(* CODESYS project connect_1.project
   Title: connect_1
   Version: 0.0.0.0
   Author: gusta

Project tree, tasks and I/O mapping:
  MyController : TM241CEC24T/U, Schneider Electric, order no. TM241CEC24T/U, version 4.0.6.18
    application Application
      libraries: Util, 3.5.1.0 (System)
      task MAST (cyclic, interval t#20ms, priority 15) calls opstart
      task Task (cyclic, interval t#5ms, priority 1) calls loop1
      task Task_1 (cyclic, interval t#20ms, priority 3) calls counter
      global variables GVL
      program opstart [ST]
      program counter [ST]
      program loop1 [ST]
      function block GPID [ST]
      program POU_1 [FBD]
    DI : Digital Inputs, Schneider Electric, version 4.0.6.18
        settings: IOs Usage = 15
        input  Application.input1 : BOOL  // IW0.I4
        input  Application.input2 : BOOL  // IW0.I5
        input  ibDI_IB1 : BYTE  // IB1
        unmapped channels: IW0
    DQ : Digital Outputs, Schneider Electric, version 4.0.6.18
        output Application.Q_enable : BOOL  // QW0.Q0
        output Application.Q_reset : BOOL  // QW0.Q1
        output Application.Q_operating : BOOL  // QW0.Q2
        output qbDQ_QB1 : BYTE  // QB1
        unmapped channels: QW0
    Counters : Counters, Schneider Electric, version 4.0.6.18
        settings: Instance name = 'HSCS'; B input History = 'old=-1 new=1'; A input History = 'old=-1 new=0'; Temporary Instance name = 'HSCS'; Instance name = 'HSCM'; B input History = 'old=-1 new=3'; A input History = 'old=-1 new=2'; Temporary Instance name = 'HSCM'
    Pulse_Generators : Pulse Generators, Schneider Electric, version 4.0.6.18
    Cartridge_1 : Cartridge, Schneider Electric, version 4.0.6.18
    IO_Bus : IO bus - TM3, Schneider Electric, version 4.0.6.18
      Module_1 : TM3AQ4/G, Schneider Electric, order no. TM3AQ4/G, version 1.0.0.12
          settings: KPI Configuration.KPI Configuration[0] = 17; KPI Configuration.KPI Configuration[1] = 17; KPI Configuration.KPI Configuration[4] = 240; KPI Configuration.KPI Configuration[5] = 216; KPI Configuration.KPI Configuration[6] = 240; KPI Configuration.KPI Configuration[7] = 216; KPI Configuration.KPI Configuration[12] = 16; KPI Configuration.KPI Configuration[13] = 39; KPI Configuration.KPI Configuration[14] = 16; KPI Configuration.KPI Configuration[15] = 39
          output qiModule_1_QW0 : INT  // QW0
          output qiModule_1_QW1 : INT  // QW1
          output qiModule_1_QW2 : INT  // QW2
          output qiModule_1_QW3 : INT  // QW3
          input  ibModule_1_IBStatusQW0 : BYTE  // IBStatusQW0
          input  ibModule_1_IBStatusQW1 : BYTE  // IBStatusQW1
          input  ibModule_1_IBStatusQW2 : BYTE  // IBStatusQW2
          input  ibModule_1_IBStatusQW3 : BYTE  // IBStatusQW3
      Module_2 : TM3SAF5R/G, Schneider Electric, order no. TM3SAF5R/G, version 1.0.1.12
          input  iwModule_2_IW0 : WORD  // IW0
          output qbModule_2_QB0 : BYTE  // QB0
    COM_Bus : COM bus, Schneider Electric, version 4.0.6.18
    Ethernet_1 : Ethernet Network, Schneider Electric, version 4.0.6.18
    Serial_Line_1 : Serial line, Schneider Electric, version 4.0.6.18
      SoMachine_Network_Manager : SoMachine-Network Manager, Schneider Electric, version 4.0.0.2
    Serial_Line_2 : Serial line, Schneider Electric, version 4.0.6.18
      Modbus_Manager : Modbus Manager, Schneider Electric, version 4.0.0.2
    CAN_1 : CANopen bus, Schneider Electric, version 4.0.6.18
  FdtConnections : FDT Connections, Schneider Electric, version 1.0.0.2
    Modbus_Serial_Line_Manager : Modbus Serial Line Manager, Schneider Electric, version 2.6.0
      Lexium_32_C : Lexium 32 C Advanced Settings, Schneider Electric, version 1.18.00.07
*)

// MyController/Application/GVL
VAR_GLOBAL
	run_loop: INT := 0;
END_VAR
VAR_GLOBAL
	test: TON;
	input2: BOOL;
	input1: BOOL;
	Q_enable: BOOL;
	Q_reset: BOOL;
	Q_operating: BOOL;
END_VAR

// MyController/Application/opstart
PROGRAM opstart
VAR
	direction: BOOL := true;
	on_startup: UINT := 1;
	timer: TON;
END_VAR


//Q7=%QX0.7
//Q8=%QX1.0
//Q9=%QX1.1
//enable = %QX12.0
//Resetmode = %QX12.1

CASE on_startup OF 
	1:
	
	Q_reset := TRUE;
	on_startup := 2;

	
	2:
	Q_reset := FALSE;
	%QX12.0 := TRUE;
	
	on_startup := 3;
	
	
	3:
	%QX12.1 := TRUE;
	on_startup := 4;
	
	4:
	%QX12.1 := FALSE;
	Q_operating := TRUE;
	IF %IX8.7 = TRUE THEN
		on_startup := 5;
		Q_reset := TRUE;
	END_IF
	
	5:
	Q_reset := FALSE;
	Q_enable := TRUE;
	on_startup := 6; 
	
	6:

	run_loop := 1;
	
	(*qiModule_1_QW0 := 1000;
	IF input2 = FALSE THEN
		Q_reset := TRUE;
		qiModule_1_QW0 := -1000;
		timer.PT := T#1000MS;
		timer.IN := TRUE;
		IF timer.Q = TRUE THEN
			qiModule_1_QW0 := -1000;
			timer.IN := FALSE;
			on_startup := 7;
			Q_reset := FALSE;
		END_IF
	END_IF
	
	
	7:
	timer.IN := TRUE;
	IF timer.Q THEN
		Q_reset := FALSE;
	END_IF*)
	
	//%QW3 := 100;
	
	(*qiModule_1_QW0 := 1000;
		IF input2 = FALSE THEN
			qiModule_1_QW0 := 0;
			Q_reset := TRUE;
			on_startup := 7;
		END_IF
		
		
	7:
		test.PT := T#4000MS;
		test.IN := TRUE;
	IF test.Q = TRUE THEN
		qiModule_1_QW0 := 0;
		test.IN := FALSE;
		Q_reset := FALSE;
		on_startup := 8;
	END_IF
		
	8:
		
		
		qiModule_1_QW0 := -1000;
	IF input1 = FALSE THEN
		qiModule_1_QW0 := 0;
		test.IN := FALSE;
		Q_reset := TRUE;
		on_startup := 9;
	END_IF
	9:
		test.PT := T#4000MS;
		test.IN := TRUE;
	IF test.Q = TRUE THEN
		qiModule_1_QW0 := 0;
		test.IN := FALSE;
		Q_reset := FALSE;
		on_startup := 6;
	END_IF
	*)
END_CASE
timer();
test();

END_PROGRAM

// MyController/Application/loop1
PROGRAM loop1
VAR
	ready: BOOL := FALSE;
	PID_theta: INT;
END_VAR
VAR
	testf: REAL := 0;
	currentDeltax: REAL := 0;
	currentTheta: REAL := 0;
	ThetaRefInput: REAL := 3.14159265359;
	PIDThetaOutput: REAL := 0;
	lastX: REAL;
	PIDTheta: PID := (KP := 19.32,TN := 1/(16.32/7.36),TV := 3.2, Y_MIN := 210, Y_MAX := 210);
	PIDXd: PD := (KP :=-0.168, TV:=0);
	PIDXcOutput: REAL;
	PIDThetaGustav: GPID := (Kp := -90.9569316890003, Ki := 1.74506598302446, Kd := 0.141819106037972, filter_C := 738.46, saturation := 210, Ti := 1, sample_T := 0.005) ;
END_VAR

IF ready THEN 
		currentTheta := Hscs.CurrentValue * 0.00613592315; // convert to radians 2*pi/1024
		currentDeltax :=  ((HSCM.CurrentValue-lastX) * 0.00001640016) / 0.005; // convert to meters from test where 0.02 is cycle time
		lastX := HSCM.CurrentValue;
(*
		//Gustav PID
		PIDThetaGustav.Ref := ThetaRefInput;
		PIDThetaGustav.input_Y := currentTheta;
		PIDThetaOutput := PIDThetaGustav.out;
		PIDThetaGustav();
		*)

		//Cart x_d controller
		PIDXd.SET_POINT := 0;
		PIDXd.ACTUAL := currentDeltax;
		PIDXd();
		PIDXcOutput := PIDXd.Y;
		//testf := PIDXcOutput; //* (2*0.72*5)/(0.034); // in Newton
		//PIDXcOutput := (PIDXcOutput)/150*10000; // correct the unit into mV
		
		//NOrmal PID
		//Theta Controller
		PIDTheta.SET_POINT := 0; //setpoint of error signal
		PIDTheta.ACTUAL := PIDXcOutput-(ThetaRefInput-currentTheta);
		PIDTheta(); // Call functionblock to update output
		PIDThetaOutput := PIDTheta.Y * (10000/210);
		
		
		//qiModule_1_QW0 := REAL_TO_INT(PIDThetaOutput);

END_IF

END_PROGRAM

// MyController/Application/GPID
FUNCTION_BLOCK GPID
VAR_INPUT
	Ref: REAL;
	input_Y: REAL;
	Kp: REAL;
	Ki: REAL;
	Kd: REAL;
	sample_T: REAL;
	filter_C: REAL;
	Ti: REAL;
END_VAR
VAR
	integral: REAL;
	until_n: REAL;
	sum: REAL;
	dif: REAL;
	filter: REAL;
	d_sum: REAL;
	differance: REAL;
	inte: REAL;
	wind_back: REAL;
	i_sum: REAL;
	anti_sum: REAL;
	integral_I: REAL;
	error: REAL := 0;
END_VAR
VAR_OUTPUT
	out: REAL;
	Y_input: REAL;
END_VAR
VAR_INPUT
	saturation: REAL;
END_VAR
VAR
	tmpOut: REAL;
END_VAR

error := ref - input_Y ;

//anti-windback


//proprtinal led
error := Kp *error;


//differance led
dif := Kd *error;
d_sum := dif - filter;
differance := filter_C *d_sum;
filter := filter + (sample_T/2)*differance;

//integral led
inte := Ki *error;

anti_sum := out - tmpOut;
wind_back := anti_sum * 1/Ti;

i_sum := inte + wind_back;
integral_I := integral_I + (sample_T/2)*i_sum; 

//sum af led
tmpOut := error + i_sum + differance; 
IF tmpOut > saturation THEN
	out := saturation;
ELSIF tmpOut < -saturation THEN 
	out := -saturation;
ELSE 
	out := tmpOut;
END_IF

END_FUNCTION_BLOCK

// MyController/Application/counter
PROGRAM counter
VAR
	temp: DINT;
	t: INT;
END_VAR


HSCS();
HSCS(EN_Enable := TRUE, EN_Preset := TRUE, F_Preset := TRUE, F_Enable := TRUE);
temp := HSCS.CurrentValue;
//HSCS();
HSCM();
HSCM.CurrentValue;
//HSCM();
	HSCM(EN_Enable := TRUE, EN_Preset := TRUE, F_Preset := TRUE, F_Enable := TRUE);

END_PROGRAM

// MyController/Application/POU_1
PROGRAM POU_1
VAR
END_VAR

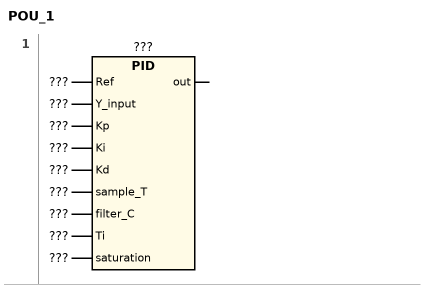
// NETWORK 1
???(); // PID

END_PROGRAM
